(* PLC project Sin nombre, Desconocido Sin nombre 1 *)
(* stored: creationDateTime 2024-10-27T15:19:01, modificationDateTime 2024-11-03T12:57:43 *)

PROGRAM lab2
  VAR
    Buzzer AT %QX0.0 : BOOL := 0;  (* Buzzer *)
    Sensor AT %IX0.0 : BOOL;  (* Sensor *)
    Boton1 AT %IX0.1 : BOOL;  (* Boton que cancela la cuenta regresiva. *)
    Boton2 AT %IX0.2 : BOOL;  (* Boton que desactiva la alarma. *)
  END_VAR
  VAR
    TON0 : TON;
    SR0 : SR;
    TP1 : TP;
    TOF0 : TOF;
    RS0 : RS;
  END_VAR

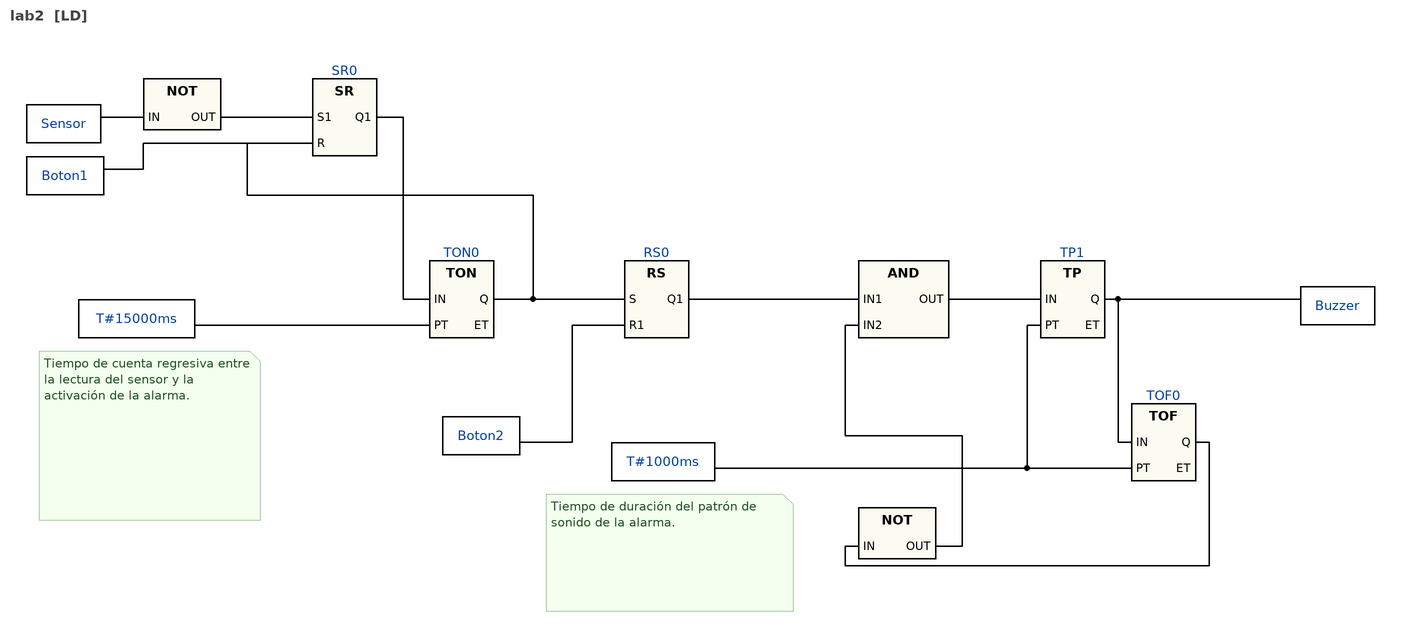
(* LD diagram, written out as Structured Text *)
SR0(S1 := NOT Sensor, R := TON0.Q OR Boton1);
TON0(IN := SR0.Q1, PT := T#15000ms);
RS0(S := TON0.Q, R1 := Boton2);
TOF0(IN := TP1.Q, PT := T#1000ms);
TP1(IN := RS0.Q1 AND NOT TOF0.Q, PT := T#1000ms);
Buzzer := TP1.Q;
(* Tiempo de cuenta regresiva entre la lectura del sensor y la activación de la alarma. *)
(* Tiempo de duración del patrón de sonido de la alarma. *)
END_PROGRAM

CONFIGURATION Config0
  RESOURCE Res0 ON PLC
    TASK task0(INTERVAL := T#20ms, PRIORITY := 0);
    PROGRAM instance0 WITH task0 : lab2;
  END_RESOURCE
END_CONFIGURATION
